{attribute 'linkalways'} 
{attribute 'no_explicit_call' := 'This FB is a CLASS and must be accessed using methods or properties'}
{attribute 'enable_dynamic_creation'}
FUNCTION_BLOCK FINAL NE_INT EXTENDS Node
VAR
	in1 : _INT(0);
	in2 : _INT(0);
	out : _BOOL(FALSE);
END_VAR

METHOD PUBLIC Clone : I_Node
VAR
	pNode : POINTER TO NE_INT;
END_VAR
pNode := __NEW(NE_INT);
Clone := pNode^;
END_METHOD

METHOD FB_init : BOOL
VAR_INPUT
	bInitRetains : BOOL; // if TRUE, the retain variables are initialized (warm start / cold start)
	bInCopyCode : BOOL;  // if TRUE, the instance afterwards gets moved into the copy code (online change)
END_VAR
AddInput('in1',THIS^.in1);
AddInput('in2',THIS^.in2);
AddOutput('out', THIS^.out);
END_METHOD

METHOD PROTECTED OnExecute
VAR
END_VAR
out.Value := in1.Value <> in2.Value;
END_METHOD

END_FUNCTION_BLOCK

(* stored: Version 1.1.0.1, ProductVersion 3.1.4024.15
   POU NE_INT: Id {d52a084a-d3aa-41e8-95d1-3a246d035606}, SpecialFunc None
   Folder Constructor: Id {5a411314-f09c-4e5f-8523-eec8ff7b6846}
   Method Clone: Id {dcd75522-aabf-4b3a-a607-3c6976e4c09a}
   Method FB_init: Id {ff2866b1-3e75-4bc1-a489-2e56d1f0887d}
   Method OnExecute: Id {ef143e41-c4ee-48d0-b94f-07329246de96} *)
